RoboDK station: 02 - Intro.rdk

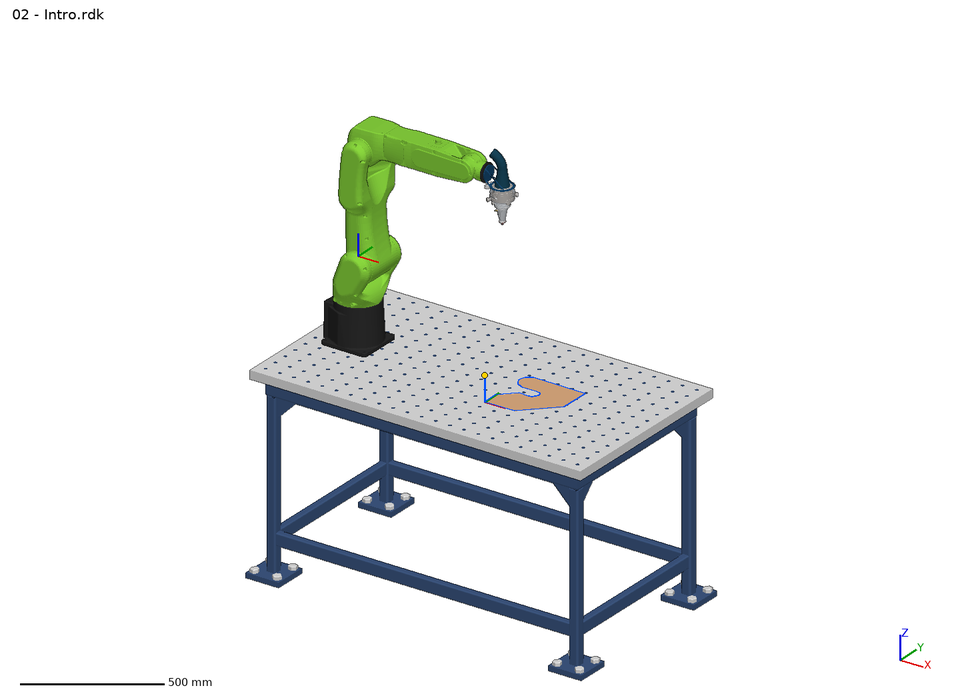
[picture v0: the station drawn from its stored meshes, robots at their saved joint values, targets as dots, program paths as lines]
Station 02 - Intro (saved by RoboDK 5.2.4). Poses are relative to the parent item; angles as X-Y-Z fixed-axis rotations.
  - frame Fanuc CR-7iA/L Base at (0, 0, 330) mm
    - robot Fanuc CR-7iA/L: 6 axes, payload 7 kg, reach 911 mm, repeatability 0.03 mm, weight 55 kg
        modified DH rows (alpha deg, a mm, theta deg, d mm): 0, 0, 0, 330; -90, 50, -90, 0; 0, 440, 0, 0; -90, 35, 0, 420; 90, 0, 0, 0; -90, 0, 0, 80
        base shift (0, 0, -330) mm
        joint limits [-170, -100, -67, -190, -115, -360] to [170, 145, 213, 190, 115, 360]; home [0, 0, 0, 0, 0, 0]; saved at [0, 0, 0, 0, 0, 0]
      - tool Cutting Head, TCP at (-183.12, 0, 59) mm, rotated rx 0 ry -90 rz 0 deg, size 285.5 x 102.9 x 112.9 mm, geometry from Cutting Head.STEP
    - frame Part at (634.18, -140.58, -330) mm
      - object Cutting sheet at (0, 0, 0) mm, size 250 x 250 x 3 mm, geometry from Cutting sheet.STEP
    - object Table 1400x800x800 at (120, 0, -330) mm, size 1420 x 820 x 800 mm, geometry from Table.sld
  - program Path1 (60 instructions, listed below)
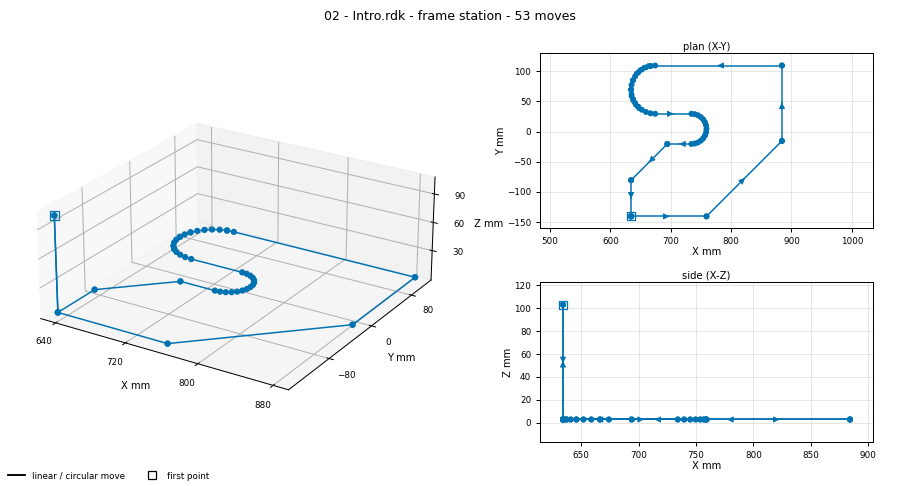
[picture p0: tool path of 02 - Intro.rdk in frame station, 53 of 53 moves have a stored position in this frame; points joined in program order, loops and branches not executed]

--- program Path1 (robot Fanuc CR-7iA/L) ---
  Smooth(1)
  Set speed (100.0 mm/s)
  Set Ref.: Frame 2 -> Part
  Set Tool: Cutting Head
  Show Cutting Head
  MoveJ 1 to (0, 0, 103) mm, rotated rx -180 ry 0 rz 0 deg; joints [-15.849, 40.1, -69.279, 16.885, 70.101, -5.898]
  MoveL 2 to (0, 0, 103) mm, rotated rx -180 ry 0 rz 0 deg; joints [-15.849, 40.1, -69.279, 16.885, 70.101, -5.898]
  MoveL 3 to (0, 0, 3) mm, rotated rx -180 ry 0 rz 0 deg; joints [-15.849, 53.371, -79.402, 16.11, 79.81, -2.925]
  MoveL 4 to (0, 0, 3) mm, rotated rx -180 ry 0 rz 0 deg; joints [-15.849, 53.371, -79.402, 16.11, 79.81, -2.925]
  Set speed (50.0 mm/s)
  MoveL 5 to (125, 0, 3) mm, rotated rx -180 ry 0 rz 0 deg; joints [-12.772, 59.496, -65.376, 14.001, 66.024, -5.786]
  MoveL 6 to (125, 0, 3) mm, rotated rx -180 ry 0 rz 0 deg; joints [-12.772, 59.496, -65.376, 14.001, 66.024, -5.786]
  MoveL 7 to (250, 125, 3) mm, rotated rx 180 ry 0 rz 0 deg; joints [-1.198, 68.044, -51.796, 1.524, 51.806, -0.943]
  MoveL 8 to (250, 125, 3) mm, rotated rx 180 ry 0 rz 0 deg; joints [-1.198, 68.044, -51.796, 1.524, 51.806, -0.943]
  MoveL 9 to (250, 250, 3) mm, rotated rx -180 ry 0 rz 0 deg; joints [8.353, 68.8, -50.729, -10.74, 51.224, 6.774]
  MoveL 10 to (250, 250, 3) mm, rotated rx -180 ry 0 rz 0 deg; joints [8.353, 68.8, -50.729, -10.74, 51.224, 6.774]
  MoveL 11 to (40, 250, 3) mm, rotated rx -180 ry 0 rz 0 deg; joints [11.555, 54.652, -75.741, -11.912, 76.036, 2.914]
  MoveL 12 to (32.2, 249.23, 3) mm, rotated rx 180 ry 0 rz 0 deg; joints [11.641, 54.314, -76.643, -11.956, 76.923, 2.743]
  MoveL 13 to (32.2, 249.23, 3) mm, rotated rx 180 ry 0 rz 0 deg; joints [11.641, 54.314, -76.643, -11.956, 76.923, 2.743]
  MoveL 14 to (24.69, 246.96, 3) mm, rotated rx -180 ry 0 rz 0 deg; joints [11.564, 53.989, -77.549, -11.835, 77.806, 2.534]
  MoveL 15 to (17.78, 243.26, 3) mm, rotated rx -180 ry 0 rz 0 deg; joints [11.319, 53.689, -78.423, -11.548, 78.651, 2.302]
  MoveL 16 to (11.72, 238.28, 3) mm, rotated rx -180 ry 0 rz 0 deg; joints [10.91, 53.426, -79.229, -11.101, 79.426, 2.062]
  MoveL 17 to (6.74, 232.22, 3) mm, rotated rx -180 ry 0 rz 0 deg; joints [10.347, 53.206, -79.933, -10.505, 80.099, 1.826]
  MoveL 18 to (3.04, 225.31, 3) mm, rotated rx 180 ry 0 rz 0 deg; joints [9.651, 53.034, -80.502, -9.783, 80.638, 1.607]
  MoveL 19 to (3.04, 225.31, 3) mm, rotated rx 180 ry 0 rz 0 deg; joints [9.651, 53.034, -80.502, -9.783, 80.638, 1.607]
  MoveL 20 to (0.77, 217.8, 3) mm, rotated rx -180 ry 0 rz 0 deg; joints [8.85, 52.916, -80.909, -8.961, 81.019, 1.41]
  MoveL 21 to (0, 210, 3) mm, rotated rx 180 ry 0 rz 0 deg; joints [7.98, 52.852, -81.134, -8.076, 81.221, 1.241]
  MoveL 22 to (0, 210, 3) mm, rotated rx 180 ry 0 rz 0 deg; joints [7.98, 52.852, -81.134, -8.076, 81.221, 1.241]
  MoveL 23 to (0.77, 202.2, 3) mm, rotated rx 180 ry 0 rz 0 deg; joints [7.082, 52.843, -81.165, -7.166, 81.233, 1.098]
  MoveL 24 to (3.04, 194.69, 3) mm, rotated rx -180 ry 0 rz 0 deg; joints [6.199, 52.89, -81, -6.275, 81.053, 0.98]
  MoveL 25 to (6.74, 187.78, 3) mm, rotated rx -180 ry 0 rz 0 deg; joints [5.372, 52.991, -80.649, -5.444, 80.69, 0.883]
  MoveL 26 to (11.72, 181.72, 3) mm, rotated rx -180 ry 0 rz 0 deg; joints [4.639, 53.146, -80.128, -4.709, 80.16, 0.806]
  MoveL 27 to (11.72, 181.72, 3) mm, rotated rx -180 ry 0 rz 0 deg; joints [4.639, 53.146, -80.128, -4.709, 80.16, 0.806]
  MoveL 28 to (17.78, 176.74, 3) mm, rotated rx -180 ry 0 rz 0 deg; joints [4.032, 53.352, -79.463, -4.101, 79.489, 0.749]
  MoveL 29 to (24.69, 173.04, 3) mm, rotated rx 180 ry 0 rz 0 deg; joints [3.573, 53.602, -78.685, -3.644, 78.707, 0.714]
  MoveL 30 to (32.2, 170.77, 3) mm, rotated rx 180 ry 0 rz 0 deg; joints [3.276, 53.891, -77.828, -3.351, 77.849, 0.706]
  MoveL 31 to (40, 170, 3) mm, rotated rx -180 ry 0 rz 0 deg; joints [3.146, 54.21, -76.929, -3.23, 76.949, 0.73]
  MoveL 32 to (100, 170, 3) mm, rotated rx -180 ry 0 rz 0 deg; joints [2.83, 57.118, -70.02, -3.011, 70.045, 1.028]
  MoveL 33 to (105.56, 169.37, 3) mm, rotated rx -180 ry 0 rz 0 deg; joints [2.744, 57.425, -69.382, -2.931, 69.407, 1.032]
  MoveL 34 to (110.85, 167.52, 3) mm, rotated rx -180 ry 0 rz 0 deg; joints [2.546, 57.72, -68.782, -2.731, 68.804, 0.988]
  MoveL 35 to (115.59, 164.55, 3) mm, rotated rx -180 ry 0 rz 0 deg; joints [2.247, 57.987, -68.249, -2.419, 68.266, 0.896]
  MoveL 36 to (119.55, 160.59, 3) mm, rotated rx 180 ry 0 rz 0 deg; joints [1.864, 58.212, -67.807, -2.013, 67.819, 0.76]
  MoveL 37 to (122.52, 155.85, 3) mm, rotated rx -180 ry 0 rz 0 deg; joints [1.416, 58.381, -67.477, -1.533, 67.484, 0.587]
  MoveL 38 to (124.37, 150.56, 3) mm, rotated rx -180 ry 0 rz 0 deg; joints [0.923, 58.486, -67.275, -1.001, 67.278, 0.387]
  MoveL 39 to (125, 145, 3) mm, rotated rx 180 ry 0 rz 0 deg; joints [0.408, 58.519, -67.209, -0.443, 67.21, 0.172]
  MoveL 40 to (124.37, 139.44, 3) mm, rotated rx 180 ry 0 rz 0 deg; joints [-0.106, 58.481, -67.284, 0.115, 67.284, -0.044]
  MoveL 41 to (122.52, 134.15, 3) mm, rotated rx 180 ry 0 rz 0 deg; joints [-0.596, 58.372, -67.495, 0.645, 67.496, -0.247]
  MoveL 42 to (119.55, 129.41, 3) mm, rotated rx 180 ry 0 rz 0 deg; joints [-1.041, 58.199, -67.833, 1.124, 67.837, -0.424]
  MoveL 43 to (115.59, 125.45, 3) mm, rotated rx 180 ry 0 rz 0 deg; joints [-1.419, 57.971, -68.281, 1.527, 68.288, -0.565]
  MoveL 44 to (110.85, 122.48, 3) mm, rotated rx 180 ry 0 rz 0 deg; joints [-1.711, 57.702, -68.82, 1.835, 68.83, -0.663]
  MoveL 45 to (105.56, 120.63, 3) mm, rotated rx -180 ry 0 rz 0 deg; joints [-1.902, 57.405, -69.424, 2.032, 69.436, -0.714]
  MoveL 46 to (100, 120, 3) mm, rotated rx 180 ry 0 rz 0 deg; joints [-1.98, 57.097, -70.063, 2.107, 70.075, -0.718]
  MoveL 47 to (60, 120, 3) mm, rotated rx -180 ry 0 rz 0 deg; joints [-2.123, 55.073, -74.667, 2.201, 74.677, -0.582]
  MoveL 48 to (60, 120, 3) mm, rotated rx -180 ry 0 rz 0 deg; joints [-2.123, 55.073, -74.667, 2.201, 74.677, -0.582]
  MoveL 49 to (0, 60, 3) mm, rotated rx -180 ry 0 rz 0 deg; joints [-9.243, 52.908, -80.937, 9.357, 81.055, -1.468]
  MoveL 50 to (0, 60, 3) mm, rotated rx -180 ry 0 rz 0 deg; joints [-9.243, 52.908, -80.937, 9.357, 81.055, -1.468]
  MoveL 51 to (0, 0, 3) mm, rotated rx -180 ry 0 rz 0 deg; joints [-15.849, 53.371, -79.402, 16.11, 79.81, -2.925]
  Set speed (100.0 mm/s)
  MoveL 52 to (0, 0, 3) mm, rotated rx -180 ry 0 rz 0 deg; joints [-15.849, 53.371, -79.402, 16.11, 79.81, -2.925]
  MoveL 53 to (0, 0, 103) mm, rotated rx -180 ry 0 rz 0 deg; joints [-15.849, 40.1, -69.279, 16.885, 70.101, -5.898]
